// SIMATIC S7-200 project (STEP 7-Micro/WIN), CPU 224XP CN REL 02.01

ORGANIZATION_BLOCK MAIN:OB1
TITLE=PROGRAM COMMENTS
BEGIN
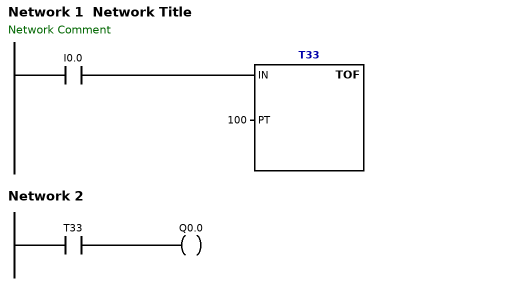
Network 1 // Network Title
// Network Comment
// (network saved uncompiled; LAD cells follow)
// row 0: c0 -| |- I0.0  c1 --  c2 [TOF T33 IN:=power@row0, PT:=100]
// row 1: c2 [box]
Network 2
LD     T33
=      Q0.0
END_ORGANIZATION_BLOCK
